// TIA Portal V15.1 export
// export: Created 2020-06-12T07:35:48.9443359Z, ExportSetting None, DisplayName Totally Integrated Automation Portal, DisplayVersion V15.1, DisplayName TIA Portal Openness, DisplayVersion V15.1, DisplayName STEP 7 Professional, DisplayVersion V15.1, DisplayName STEP 7 Safety, DisplayVersion V15.1, DisplayName WinCC Advanced, DisplayVersion V15.1
FUNCTION "XY_move" : Void   // FC801, FBD
TITLE = ESM XY-shift
{ S7_Optimized_Access := 'FALSE' }
// stored: SetENOAutomatically False
   VAR_TEMP
      tcsf : Bool;
      tlock_rgt : Bool;
      tlock_lft : Bool;
      tlock_fwd : Bool;
      tlock_bwd : Bool;
      tlock_melt : Bool;
      tmove_cmd : Bool;
      tlock_ext : Bool;
      tQ1 : Bool;
      tQ2 : Bool;
      tQ3 : Bool;
      tBypass : Bool;
      tBool : Bool;
      tPosX : Real;
      tPosY : Real;
      tCmdLeft : Bool;
      tCmdRight : Bool;
      tCmdFwd : Bool;
      tCmdBwd : Bool;
      tCmdCenter : Bool;
      tCmdEn : Bool;
   END_VAR
BEGIN

REGION Network 1: common system fault
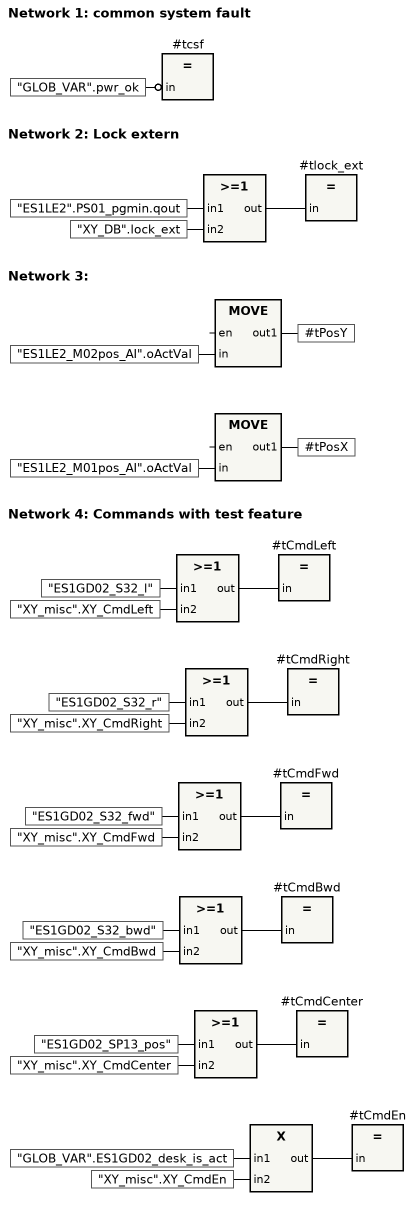
   #tcsf := NOT "GLOB_VAR".pwr_ok;
END_REGION

REGION Network 2: Lock extern
   #tlock_ext := "ES1LE2".PS01_pgmin.qout OR "XY_DB".lock_ext;
END_REGION

REGION Network 3
   #tPosY := "ES1LE2_M02pos_AI".oActVal;
   #tPosX := "ES1LE2_M01pos_AI".oActVal;
END_REGION

REGION Network 4: Commands with test feature
   #tCmdLeft := "ES1GD02_S32_l" OR "XY_misc".XY_CmdLeft;
   #tCmdRight := "ES1GD02_S32_r" OR "XY_misc".XY_CmdRight;
   #tCmdFwd := "ES1GD02_S32_fwd" OR "XY_misc".XY_CmdFwd;
   #tCmdBwd := "ES1GD02_S32_bwd" OR "XY_misc".XY_CmdBwd;
   #tCmdCenter := "ES1GD02_SP13_pos" OR "XY_misc".XY_CmdCenter;
   #tCmdEn := "GLOB_VAR".ES1GD02_desk_is_act XOR "XY_misc".XY_CmdEn;
END_REGION

REGION Network 5: Call Funktionblock XY Move
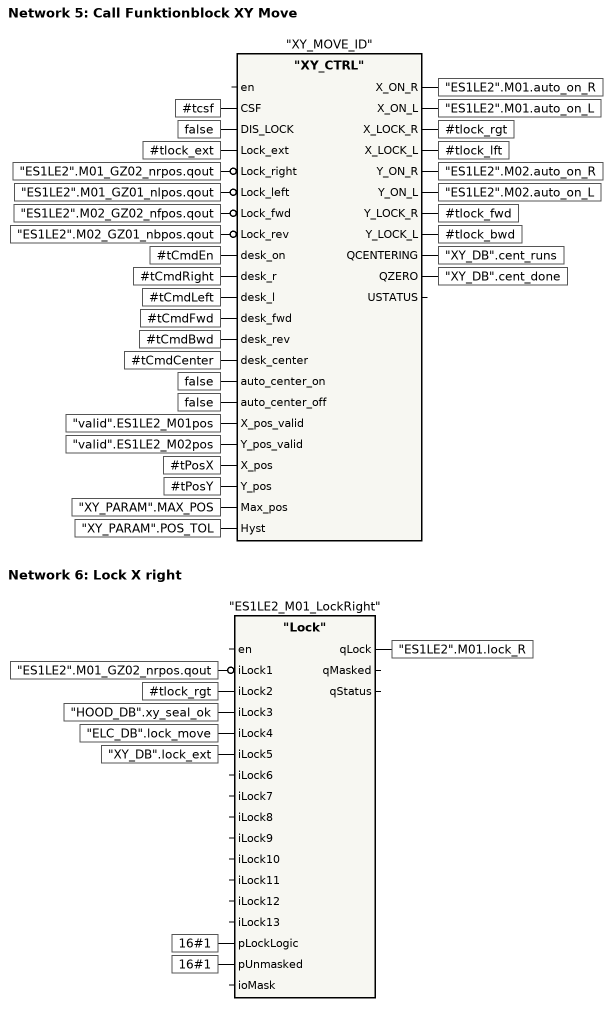
   "XY_MOVE_ID"(CSF := #tcsf,   // "XY_CTRL"
                DIS_LOCK := false,
                Lock_ext := #tlock_ext,
                Lock_right := NOT "ES1LE2".M01_GZ02_nrpos.qout,
                Lock_left := NOT "ES1LE2".M01_GZ01_nlpos.qout,
                Lock_fwd := NOT "ES1LE2".M02_GZ02_nfpos.qout,
                Lock_rev := NOT "ES1LE2".M02_GZ01_nbpos.qout,
                desk_on := #tCmdEn,
                desk_r := #tCmdRight,
                desk_l := #tCmdLeft,
                desk_fwd := #tCmdFwd,
                desk_rev := #tCmdBwd,
                desk_center := #tCmdCenter,
                auto_center_on := false,
                auto_center_off := false,
                X_pos_valid := "valid".ES1LE2_M01pos,
                Y_pos_valid := "valid".ES1LE2_M02pos,
                X_pos := #tPosX,
                Y_pos := #tPosY,
                Max_pos := "XY_PARAM".MAX_POS,
                Hyst := "XY_PARAM".POS_TOL,
                X_ON_R => "ES1LE2".M01.auto_on_R,
                X_ON_L => "ES1LE2".M01.auto_on_L,
                X_LOCK_R => #tlock_rgt,
                X_LOCK_L => #tlock_lft,
                Y_ON_R => "ES1LE2".M02.auto_on_R,
                Y_ON_L => "ES1LE2".M02.auto_on_L,
                Y_LOCK_R => #tlock_fwd,
                Y_LOCK_L => #tlock_bwd,
                QCENTERING => "XY_DB".cent_runs,
                QZERO => "XY_DB".cent_done);
END_REGION

REGION Network 6: Lock X right
   "ES1LE2_M01_LockRight"(iLock1 := NOT "ES1LE2".M01_GZ02_nrpos.qout,   // "Lock"
                          iLock2 := #tlock_rgt,
                          iLock3 := "HOOD_DB".xy_seal_ok,
                          iLock4 := "ELC_DB".lock_move,
                          iLock5 := "XY_DB".lock_ext,
                          pLockLogic := 16#1,
                          pUnmasked := 16#1,
                          qLock => "ES1LE2".M01.lock_R);
END_REGION

REGION Network 7: Lock X left
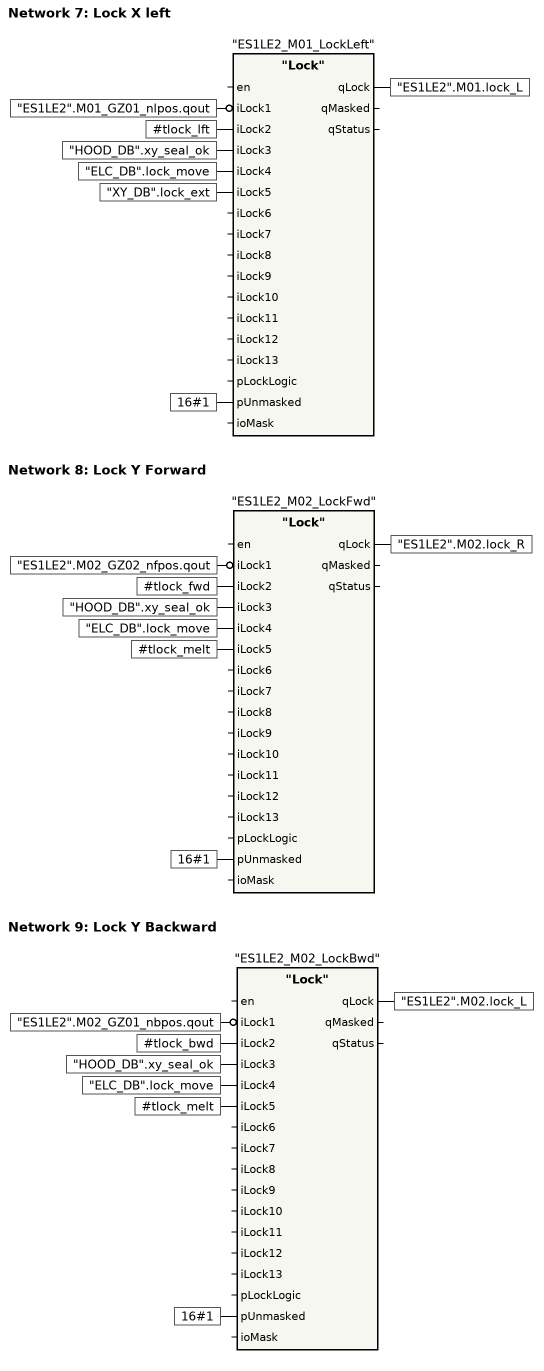
   "ES1LE2_M01_LockLeft"(iLock1 := NOT "ES1LE2".M01_GZ01_nlpos.qout,   // "Lock"
                         iLock2 := #tlock_lft,
                         iLock3 := "HOOD_DB".xy_seal_ok,
                         iLock4 := "ELC_DB".lock_move,
                         iLock5 := "XY_DB".lock_ext,
                         pUnmasked := 16#1,
                         qLock => "ES1LE2".M01.lock_L);
END_REGION

REGION Network 8: Lock Y Forward
   "ES1LE2_M02_LockFwd"(iLock1 := NOT "ES1LE2".M02_GZ02_nfpos.qout,   // "Lock"
                        iLock2 := #tlock_fwd,
                        iLock3 := "HOOD_DB".xy_seal_ok,
                        iLock4 := "ELC_DB".lock_move,
                        iLock5 := #tlock_melt,
                        pUnmasked := 16#1,
                        qLock => "ES1LE2".M02.lock_R);
END_REGION

REGION Network 9: Lock Y Backward
   "ES1LE2_M02_LockBwd"(iLock1 := NOT "ES1LE2".M02_GZ01_nbpos.qout,   // "Lock"
                        iLock2 := #tlock_bwd,
                        iLock3 := "HOOD_DB".xy_seal_ok,
                        iLock4 := "ELC_DB".lock_move,
                        iLock5 := #tlock_melt,
                        pUnmasked := 16#1,
                        qLock => "ES1LE2".M02.lock_L);
END_REGION

REGION Network 10: Hardwarelock M01 Right
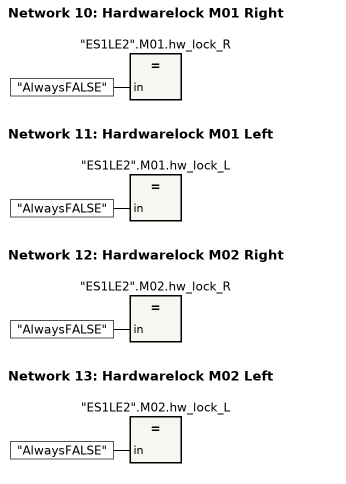
   "ES1LE2".M01.hw_lock_R := "AlwaysFALSE";
END_REGION

REGION Network 11: Hardwarelock M01 Left
   "ES1LE2".M01.hw_lock_L := "AlwaysFALSE";
END_REGION

REGION Network 12: Hardwarelock M02 Right
   "ES1LE2".M02.hw_lock_R := "AlwaysFALSE";
END_REGION

REGION Network 13: Hardwarelock M02 Left
   "ES1LE2".M02.hw_lock_L := "AlwaysFALSE";
END_REGION
END_FUNCTION
